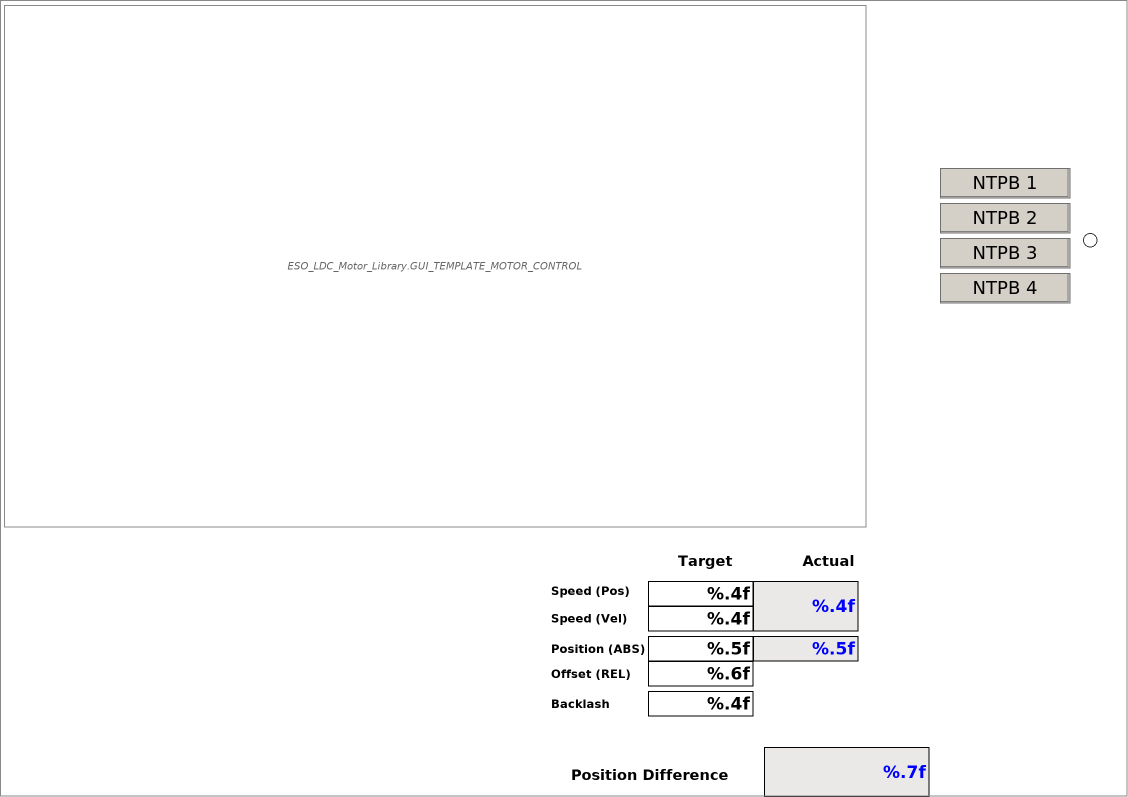
VISUALIZATION GUI_NOTT_TIP_B_CTRL  // 1128x797
    Frame (4,5 862x522)
        shows ESO_LDC_Motor_Library.GUI_TEMPLATE_MOTOR_CONTROL(m_Instance := MAIN.nott_ics.TipTilt.ptrTipActuatorsB[MAIN.nott_ics.TipTilt.guiTipActuatorsBIndex]^)
    Rectangle (548,581 95x20), "Speed (Pos)"
    Rectangle (753,636 105x25), "%.5f", text variable: MAIN.nott_ics.Delay_Lines.ptrDelayLines[MAIN.nott_ics.Delay_Lines.guiShutterIndex]^.stat.lrPosActual, input disabled if: false
    Rectangle (675,551 190x20), "Target Actual"
    Rectangle (548,639 95x20), "Position (ABS)"
    Rectangle (753,581 105x50), "%.4f", text variable: MAIN.nott_ics.Delay_Lines.ptrDelayLines[MAIN.nott_ics.Delay_Lines.guiShutterIndex]^.stat.lrVelActual, input disabled if: false
    Rectangle (648,606 105x25), "%.4f", text variable: MAIN.nott_ics.Delay_Lines.ptrDelayLines[MAIN.nott_ics.Delay_Lines.guiShutterIndex]^.ctrl.lrVelocity
        OnMouseDown: write the text variable via Default
    Rectangle (548,694 95x20), "Backlash"
    Rectangle (648,691 105x25), "%.4f", text variable: MAIN.nott_ics.Delay_Lines.ptrDelayLines[MAIN.nott_ics.Delay_Lines.guiShutterIndex]^.cfg.lrBacklash
        OnMouseDown: write the text variable via Default
    Rectangle (548,606 95x25), "Speed (Vel)"
    Rectangle (648,636 105x25), "%.5f", tooltip "Absolute position used by "MOVE ABS"", text variable: MAIN.nott_ics.Delay_Lines.ptrDelayLines[MAIN.nott_ics.Delay_Lines.guiShutterIndex]^.ctrl.lrPosition
        OnMouseDown: write the text variable via Default
    Rectangle (648,581 105x25), "%.4f", text variable: MAIN.nott_ics.Delay_Lines.ptrDelayLines[MAIN.nott_ics.Delay_Lines.guiShutterIndex]^.cfg.lrDefaultVelocity
        OnMouseDown: write the text variable via Default
    Rectangle (548,664 95x20), "Offset (REL)"
    Rectangle (648,661 105x25), "%.6f", tooltip "Relative offset used by "MOVE REL"", text variable: MAIN.nott_ics.Delay_Lines.ptrDelayLines[MAIN.nott_ics.Delay_Lines.guiShutterIndex]^.ctrl.lrOffset
        OnMouseDown: write the text variable via Default
    Rectangle (764,747 165x50), "%.7f", text variable: MAIN.nott_ics.Delay_Lines.ptrDelayLines[MAIN.nott_ics.Delay_Lines.guiShutterIndex]^.stat.lrPosError, input disabled if: false
    Rectangle (568,765 190x20), "Position Difference"
    RadioButton (1081,170 47x140), variable: MAIN.nott_ics.TipTilt.guiTipActuatorsBIndex-1
        Areas[0]: Text=Radiobutton
        Areas[1]: Text=Radiobutton
    Button (940,168 130x30), "NTPB 1"
        OnMouseClick: execute { MAIN.nott_ics.TipTilt.guiTipActuatorsBIndex := 1; }
    Button (940,203 130x30), "NTPB 2"
        OnMouseClick: execute { MAIN.nott_ics.TipTilt.guiTipActuatorsBIndex := 2; }
    Button (940,238 130x30), "NTPB 3"
        OnMouseClick: execute { MAIN.nott_ics.TipTilt.guiTipActuatorsBIndex := 3; }
    Button (940,273 130x30), "NTPB 4"
        OnMouseClick: execute { MAIN.nott_ics.TipTilt.guiTipActuatorsBIndex := 4; }
END_VISUALIZATION

(* stored: Version 1.1.0.1, ProductVersion 3.1.4024.12
   Visu GUI_NOTT_TIP_B_CTRL: Id {8b593c5a-b54c-4777-8c28-eb938c4c4e60} *)
